// Mitsubishi GX Works2 project: lednhapnhaytest   PLC: Q03UDE

PROGRAM MAIN
VAR
  ssbt : BOOL;
  ledd1 : BOOL;
  ledd2 : BOOL;
  stopbt : BOOL;
  estopbt : BOOL;
END_VAR
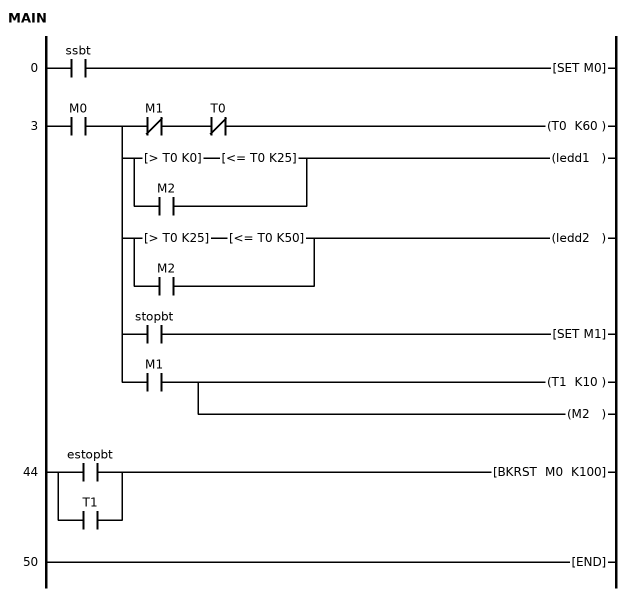
0     LD      ssbt
      SET     M0
3     LD      M0
      MPS
      ANI     M1
      ANI     T0
      OUT     T0 K60
      MRD
      LD>     T0 K0
      AND<=   T0 K25
      OR      M2
      ANB
      OUT     ledd1
      MRD
      LD>     T0 K25
      AND<=   T0 K50
      OR      M2
      ANB
      OUT     ledd2
      MRD
      AND     stopbt
      SET     M1
      MPP
      AND     M1
      OUT     T1 K10
      OUT     M2
44    LD      estopbt
      OR      T1
      BKRST   M0 K100
50    END
END_PROGRAM
